Universal Robots PolyScope program: interpreter_mode.urp

Program interpreter_mode (installation=default directory=/programs createdIn=5.10.0 lastSavedIn=5.13.1 robotSerialNumber=20215300223)
Calibrated DH parameters: a=[-0.000161, -0.235904, -0.090943, 0.0001, -0.000132, 0]; d=[0.151746, 53.298129, 72.418109, -125.585258, 0.085393, 0.092182]; alpha=[1.570518, 0.001152, 0.001536, 1.571994, -1.571888, 0]; deltaTheta=[0, 0.254593, 7.159278, -1.130689, 0.000001, 0]
InitVariablesNode
Robot Program (runOnlyOnce=true)
  Script: global exit_thread = False
  Script: interpreter_mode(clearOnEnd = False)
  Script: interpreter_mode()
